FUNCTION_BLOCK TimeOut (* Composite Function Block Type *)
  (* Standard: 61499-2 *)
  (* Version 0.0, 7/17/2026, Schneider Electric, template *)
  PACKAGE SE.Nereda;
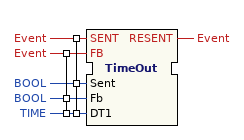
  EVENT_INPUT
    SENT WITH Sent, DT1; (* Initialization Request *)
    FB WITH Fb, DT1; (* Normal Execution Request *)
  END_EVENT
  EVENT_OUTPUT
    RESENT; (* Execution Confirmation *)
  END_EVENT
  VAR_INPUT
    Sent : BOOL;
    Fb : BOOL;
    DT1 : TIME; (* Delay Time *)
  END_VAR
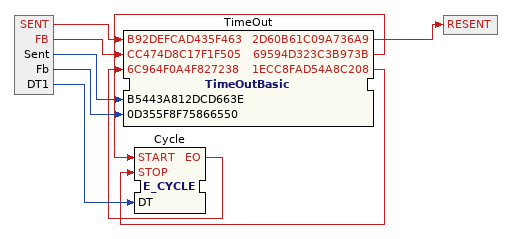
  FBS
    TimeOut : TimeOutBasic;
    Cycle : E_CYCLE;
  END_FBS
  EVENT_CONNECTIONS
    SENT TO TimeOut.B92DEFCAD435F463;
    FB TO TimeOut.CC474D8C17F1F505;
    TimeOut.2D60B61C09A736A9 TO RESENT;
    TimeOut.69594D323C3B973B TO Cycle.START;
    Cycle.EO TO TimeOut.6C964F0A4F827238;
    TimeOut.1ECC8FAD54A8C208 TO Cycle.STOP;
  END_CONNECTIONS
  DATA_CONNECTIONS
    Sent TO TimeOut.B5443A812DCD663E;
    Fb TO TimeOut.0D355F8F75866550;
    DT1 TO Cycle.DT;
  END_CONNECTIONS
END_FUNCTION_BLOCK
